// Implicitly generated code : DO NOT EDIT
FUNCTION CheckPointer : POINTER TO BYTE
VAR_INPUT 
	ptToTest : POINTER TO BYTE; // Destination address of the pointer
	iSize : DINT;		        // Size of the type the pointer points to. (e.g: 20 for POINTER TO ARRAY [0..9] OF INT) 
	iGran : DINT;		        // Granularity of the pointer access. This is the size of the biggest non-structured data type in the type the pointer points to. (e.g: 2 for POINTER TO ARRAY [0..9] OF INT)
	bWrite: BOOL;		        // Indicates read or write Access. TRUE = write access.
END_VAR

// No standard way of implementation. Fill your own code here
CheckPointer := ptToTest;

END_FUNCTION

(* stored: Version 1.1.0.1, ProductVersion 3.1.4026.13, FileIdentifier 8201619f9e1a5bf412e68bdd600ffd9d8c3452ed, FileSignature 82984454928b2e7455c487a906874577991fc4771b7159858e4784914b463eebe5394f69328c0063a2001eb8e3c4c3dd8cb7a60c881d804f7c6d902571b88019629246858fdec0ba7e292b3a3b8d86cd1f3cb34009c2713787dc8f4d3a55dfe71c82c7212748b984a9f9e865f90ab9febc416b308a445ff5a75033d973b5bb61f43f91c12f040ff2c43ba081f3ef075ff36828aea9a1400bc2f682d5bbb8280a13cf1fa2d3a55ed67d7519dad0780e08253e8a7474ef9fb5deb9f24dca4d1c9670a82dbf28be811049151af1406db89476e3b8448fdfa286e7a8b18273a4fafff88a0daf66160ee96b9b178cc0c87675698c856076fc2c267e2e9baaeffe8e0e
   POU CheckPointer: Id {3895abb6-6bea-415e-aa19-6145889f9d6e}, SpecialFunc CheckPointer *)
